PROGRAM MAIN
VAR
END_VAR

PrgMqttCom();

END_PROGRAM

(* stored: Version 1.1.0.1, ProductVersion 3.1.4022.18
   POU MAIN: Id {4325d483-c02f-4708-af5c-2f36e52f8768}, SpecialFunc None *)
